Yaskawa INFORM job: CYLINDER1.JBI

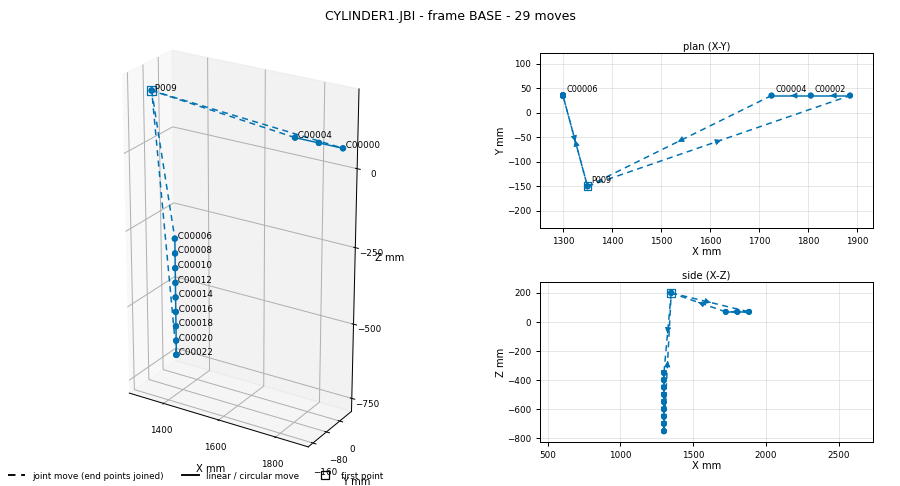
[picture p0: tool path of CYLINDER1.JBI in frame BASE, 29 of 29 moves have a stored position in this frame; points joined in program order, loops and branches not executed]
/JOB
//NAME CYLINDER1
//POS
///NPOS 26,0,26,1,0,1
///TOOL 0
///POSTYPE BASE
///RECTAN
///RCONF 0,0,0,0,0,0,0,0,0,0,0,0,0,0,0,0,0,0,0,0,0,0,0,0
C00000=1885.000,35.000,70.000,-178.0000,0.0000,0.0000
C00001=1885.000,35.000,70.000,-178.0000,0.0000,0.0000
C00002=1805.000,35.000,70.000,-178.0000,0.0000,0.0000
C00003=1805.000,35.000,70.000,-178.0000,0.0000,0.0000
C00004=1725.000,35.000,70.000,-178.0000,0.0000,0.0000
C00005=1725.000,35.000,70.000,-178.0000,0.0000,0.0000
C00006=1300.000,35.000,-350.000,-180.0000,-90.0000,0.0000
C00007=1300.000,35.000,-350.000,-180.0000,-90.0000,0.0000
C00008=1300.000,35.000,-400.000,-180.0000,-90.0000,0.0000
C00009=1300.000,35.000,-400.000,-180.0000,-90.0000,0.0000
C00010=1300.000,35.000,-450.000,-180.0000,-90.0000,0.0000
C00011=1300.000,35.000,-450.000,-180.0000,-90.0000,0.0000
C00012=1300.000,35.000,-500.000,-180.0000,-90.0000,0.0000
C00013=1300.000,35.000,-500.000,-180.0000,-90.0000,0.0000
C00014=1300.000,35.000,-550.000,-180.0000,-90.0000,0.0000
C00015=1300.000,35.000,-550.000,-180.0000,-90.0000,0.0000
C00016=1300.000,35.000,-600.000,-180.0000,-90.0000,0.0000
C00017=1300.000,35.000,-600.000,-180.0000,-90.0000,0.0000
C00018=1300.000,35.000,-650.000,-180.0000,-90.0000,0.0000
C00019=1300.000,35.000,-650.000,-180.0000,-90.0000,0.0000
C00020=1300.000,35.000,-700.000,-180.0000,-90.0000,0.0000
C00021=1300.000,35.000,-700.000,-180.0000,-90.0000,0.0000
C00022=1300.000,35.000,-750.000,-180.0000,-90.0000,0.0000
C00023=1300.000,35.000,-750.000,-180.0000,-90.0000,0.0000
C00024=1300.000,35.000,-750.000,-180.0000,-70.0000,0.0000
C00025=1300.000,35.000,-750.000,-180.0000,-70.0000,0.0000
///POSTYPE PULSE
///PULSE
EC00000=0
EC00001=368640
EC00002=368640
EC00003=0
EC00004=0
EC00005=368640
EC00006=368640
EC00007=0
EC00008=0
EC00009=368640
EC00010=368640
EC00011=0
EC00012=0
EC00013=368640
EC00014=368640
EC00015=0
EC00016=0
EC00017=368640
EC00018=368640
EC00019=0
EC00020=0
EC00021=368640
EC00022=368640
EC00023=0
EC00024=0
EC00025=368640
///POSTYPE BASE
///RECTAN
///RCONF 1,0,0,0,0,0,0,0,0,0,0,0,0,0,0,0,0,0,0,0,0,0,0,0
P00009=1350.000,-150.000,200.000,-180.0000,-45.0000,0.0000
///POSTYPE PULSE
///PULSE
EX00000=0
//INST
///DATE 2023/02/09 11:49
///ATTR SC,RW,RJ
////FRAME BASE
///GROUP1 RB1,ST1
NOP
MOVJ P009 EX000 VJ=15.00
MOVJ C00000 EC00000 VJ=10.00
CALL JOB:SPYON
MOVJ C00001 EC00001 VJ=10.00
MOVL C00002 EC00002 V=150.0
MOVJ C00003 EC00003 VJ=10.00
MOVL C00004 EC00004 V=150.0
MOVJ C00005 EC00005 VJ=10.00
CALL JOB:SPYOF
MOVJ P009 VJ=15.00
MOVJ C00006 EC00006 VJ=15.00
CALL JOB:SPYON
MOVJ C00007 EC00007 VJ=10.00
MOVL C00008 EC00008 V=150.0
MOVJ C00009 EC00009 VJ=10.00
MOVL C00010 EC00010 V=150.0
MOVJ C00011 EC00011 VJ=10.00
MOVL C00012 EC00012 V=150.0
MOVJ C00013 EC00013 VJ=10.00
MOVL C00014 EC00014 V=150.0
MOVJ C00015 EC00015 VJ=10.00
MOVL C00016 EC00016 V=150.0
MOVJ C00017 EC00017 VJ=10.00
MOVL C00018 EC00018 V=150.0
MOVJ C00019 EC00019 VJ=10.00
MOVL C00020 EC00020 V=150.0
MOVJ C00021 EC00021 VJ=10.00
MOVL C00022 EC00022 V=150.0
MOVJ C00023 EC00023 VJ=10.00
MOVL C00024 EC00024 V=150.0
MOVJ C00025 EC00025 VJ=10.00
CALL JOB:SPYOF
MOVJ P009 EX000 VJ=15.00
END
